PROGRAM TimeOptimizeCtrl
VAR
(************************ MinMax Declaration  *********************************************************************************)
	fbV2MasterTimeBlockWithMinMax: fbV2_MasterTimeBlockWithMinMax;
	LDBasketInfo: DSV2_BasketInfo;

	AR3SiSortedMTBFreeArm_Scanning				: ARRAY[1..iArmQty, 1..iMasterBlockQty, 1..3] OF INT;
	AR3SiSortedMTBFreeStn_Scanning				: ARRAY[1..iStnQty, 1..iMasterBlockQty, 1..3] OF INT;
	AR3SiSortedMTBFreeUld_Scanning				: ARRAY[1..iUldStnQty, 1..iMasterBlockQty, 1..3] OF INT;
	ARiMTBFreeSlotDataQtyArm_Scanning			: ARRAY[1..iArmQty] OF INT;
	ARiMTBFreeSlotDataQtyStn_Scanning			: ARRAY[1..iStnQty] OF INT;
	ARiMTBFreeSlotDataQtyUld_Scanning			: ARRAY[1..iUldStnQty] OF INT;

	bScanBusyFlag						: BOOL;

	diSinceStartRunningTime					: DINT;
	diSinceCopyRunningTime					: DINT;
	iCheckStep								: INT;
	bAutoRetry								: BOOL;
	tAutoRetryTimerEV						: TIME;



(************************ MinMax Declaration END *********************************************************************************)



	DelayTime: TIME := t#1s;
	TON2: TON;
	LdPnpStRE: R_TRIG;
	LdPnpStFE: F_TRIG;



	bManualRecipeGenerateEN: BOOL;
(*	fbV2SubMTBFreeSlotGenerator: fbV2_SubMTBFreeSlotGenerator;*)
	MTB_ArmTimeOK: BOOL;
	ArmPnpStep3: BOOL;
	bArmPnpStep3: BOOL;
	bArmPnpStep5: BOOL;
END_VAR

VAR PERSISTENT

	AR2SiManualSimulationInput : ARRAY [1..iRecipeBlockQty, 1..2] OF INT;  (*1st Array=Steps 	2nd Array[1]=ProcessTime/ArmTransferTime 	2ndArray[2]=StnID*)
(*	AR2SiManualRecipeTimeBlockNoCallArmTime : ARRAY[1..iRecipeBlockQty, 1..3] OF INT;
	AR2SiManualRecipeTimeBlockWithCallArmTime : ARRAY[1..iRecipeBlockQty, 1..3] OF INT;
*)

(*	bSMTBFSG: BOOL;
	bBusy: BOOL;
	bDone : BOOL;
	ARiFreeSlotDataQtyArm									: ARRAY[1..iArmQty] OF INT;
	ARiFreeSlotDataQtyStn									: ARRAY[1..iStnQty] OF INT;
	ARiFreeSlotDataQtyUld									: ARRAY[1..iUldStnQty] OF INT;


	AR3SiMasterTimeBlockFreeArm_MTB		 			: ARRAY[1..iArmQty, 1..iMasterBlockQty, 1..3] OF INT;
	AR3SiMasterTimeBlockFreeStn_MTB					: ARRAY[1..iStnQty, 1..iMasterBlockQty, 1..3] OF INT;
	AR3SiMasterTimeBlockFreeUld_MTB					: ARRAY[1..iUldStnQty, 1..iMasterBlockQty, 1..3] OF INT;
*)
END_VAR

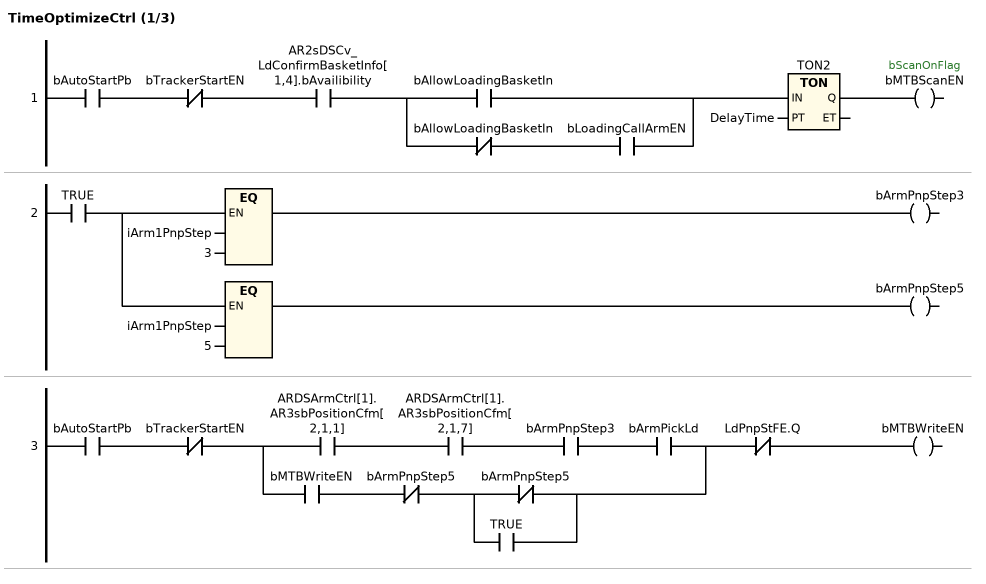
// NETWORK 1
//   bMTBScanEN: bScanOnFlag
TON2(IN := bAutoStartPb AND NOT bTrackerStartEN AND AR2sDSCv_LdConfirmBasketInfo[1,4].bAvailibility AND (bAllowLoadingBasketIn OR NOT bAllowLoadingBasketIn AND bLoadingCallArmEN), PT := DelayTime); // TON
bMTBScanEN := TON2.Q;

// NETWORK 2
bArmPnpStep3 := iArm1PnpStep = 3;
bArmPnpStep5 := iArm1PnpStep = 5;

// NETWORK 3
bMTBWriteEN := (bAutoStartPb AND NOT bTrackerStartEN AND (ARDSArmCtrl[1].AR3sbPositionCfm[2,1,1] AND ARDSArmCtrl[1].AR3sbPositionCfm[2,1,7] AND bArmPnpStep3 AND bArmPickLd OR bMTBWriteEN AND NOT bArmPnpStep5 AND (NOT bArmPnpStep5 OR TRUE))) AND NOT LdPnpStFE.Q;

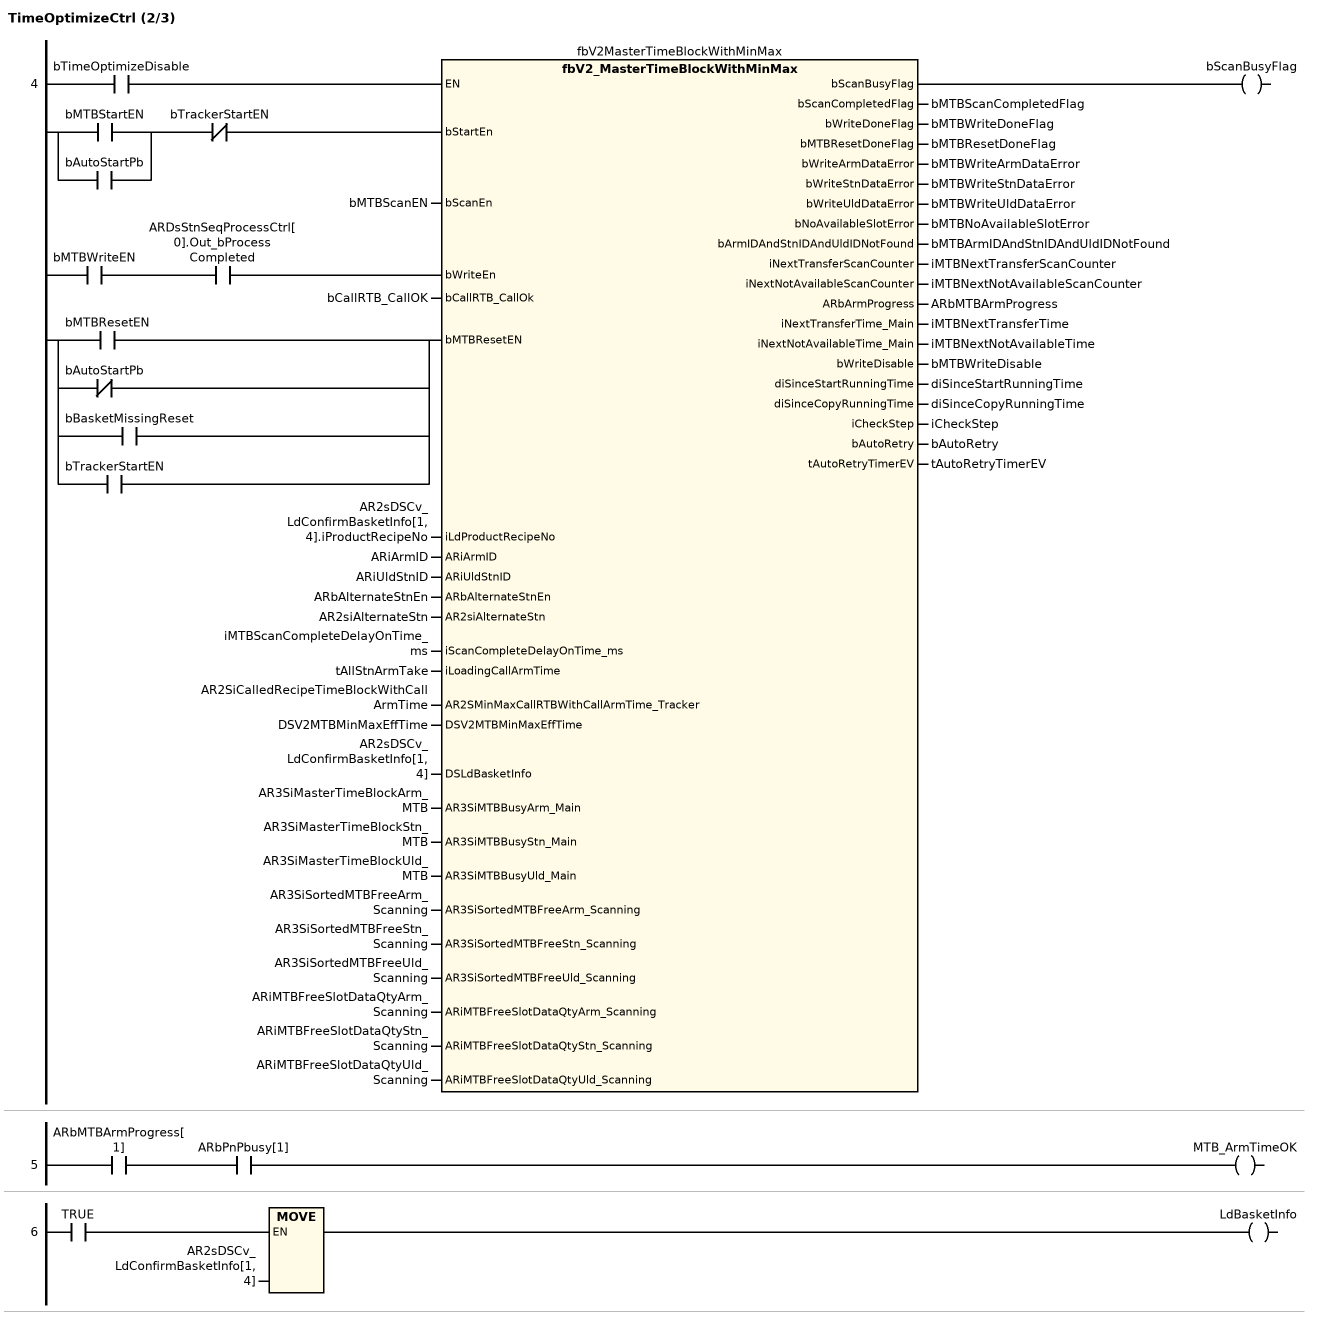
// NETWORK 4
IF bTimeOptimizeDisable THEN
    fbV2MasterTimeBlockWithMinMax(
        bStartEn := (bMTBStartEN OR bAutoStartPb) AND NOT bTrackerStartEN,
        bScanEn := bMTBScanEN,
        bWriteEn := bMTBWriteEN AND ARDsStnSeqProcessCtrl[0].Out_bProcessCompleted,
        bCallRTB_CallOk := bCallRTB_CallOK,
        bMTBResetEN := bMTBResetEN OR NOT bAutoStartPb OR bBasketMissingReset OR bTrackerStartEN,
        iLdProductRecipeNo := AR2sDSCv_LdConfirmBasketInfo[1,4].iProductRecipeNo,
        ARiArmID := ARiArmID,
        ARiUldStnID := ARiUldStnID,
        ARbAlternateStnEn := ARbAlternateStnEn,
        AR2siAlternateStn := AR2siAlternateStn,
        iScanCompleteDelayOnTime_ms := iMTBScanCompleteDelayOnTime_ms,
        iLoadingCallArmTime := tAllStnArmTake,
        AR2SMinMaxCallRTBWithCallArmTime_Tracker := AR2SiCalledRecipeTimeBlockWithCallArmTime,
        DSV2MTBMinMaxEffTime := DSV2MTBMinMaxEffTime,
        DSLdBasketInfo := AR2sDSCv_LdConfirmBasketInfo[1,4],
        AR3SiMTBBusyArm_Main := AR3SiMasterTimeBlockArm_MTB,
        AR3SiMTBBusyStn_Main := AR3SiMasterTimeBlockStn_MTB,
        AR3SiMTBBusyUld_Main := AR3SiMasterTimeBlockUld_MTB,
        AR3SiSortedMTBFreeArm_Scanning := AR3SiSortedMTBFreeArm_Scanning,
        AR3SiSortedMTBFreeStn_Scanning := AR3SiSortedMTBFreeStn_Scanning,
        AR3SiSortedMTBFreeUld_Scanning := AR3SiSortedMTBFreeUld_Scanning,
        ARiMTBFreeSlotDataQtyArm_Scanning := ARiMTBFreeSlotDataQtyArm_Scanning,
        ARiMTBFreeSlotDataQtyStn_Scanning := ARiMTBFreeSlotDataQtyStn_Scanning,
        ARiMTBFreeSlotDataQtyUld_Scanning := ARiMTBFreeSlotDataQtyUld_Scanning,
        bScanCompletedFlag => bMTBScanCompletedFlag,
        bWriteDoneFlag => bMTBWriteDoneFlag,
        bMTBResetDoneFlag => bMTBResetDoneFlag,
        bWriteArmDataError => bMTBWriteArmDataError,
        bWriteStnDataError => bMTBWriteStnDataError,
        bWriteUldDataError => bMTBWriteUldDataError,
        bNoAvailableSlotError => bMTBNoAvailableSlotError,
        bArmIDAndStnIDAndUldIDNotFound => bMTBArmIDAndStnIDAndUldIDNotFound,
        iNextTransferScanCounter => iMTBNextTransferScanCounter,
        iNextNotAvailableScanCounter => iMTBNextNotAvailableScanCounter,
        ARbArmProgress => ARbMTBArmProgress,
        iNextTransferTime_Main => iMTBNextTransferTime,
        iNextNotAvailableTime_Main => iMTBNextNotAvailableTime,
        bWriteDisable => bMTBWriteDisable,
        diSinceStartRunningTime => diSinceStartRunningTime,
        diSinceCopyRunningTime => diSinceCopyRunningTime,
        iCheckStep => iCheckStep,
        bAutoRetry => bAutoRetry,
        tAutoRetryTimerEV => tAutoRetryTimerEV); // fbV2_MasterTimeBlockWithMinMax
END_IF
bScanBusyFlag := fbV2MasterTimeBlockWithMinMax.bScanBusyFlag;

// NETWORK 5
MTB_ArmTimeOK := ARbMTBArmProgress[1] AND ARbPnPbusy[1];

// NETWORK 6
LdBasketInfo := AR2sDSCv_LdConfirmBasketInfo[1,4];

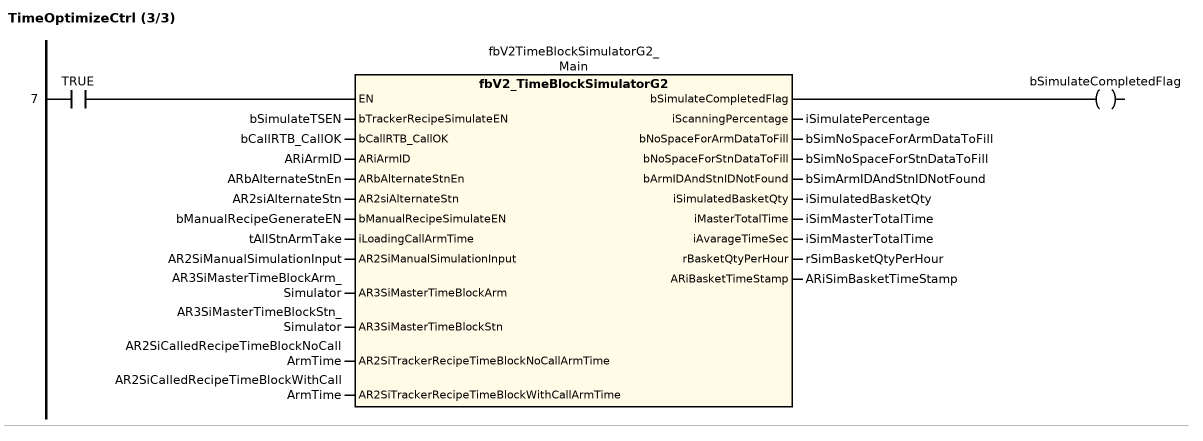
// NETWORK 7
fbV2TimeBlockSimulatorG2_Main(
    bTrackerRecipeSimulateEN := bSimulateTSEN,
    bCallRTB_CallOK := bCallRTB_CallOK,
    ARiArmID := ARiArmID,
    ARbAlternateStnEn := ARbAlternateStnEn,
    AR2siAlternateStn := AR2siAlternateStn,
    bManualRecipeSimulateEN := bManualRecipeGenerateEN,
    iLoadingCallArmTime := tAllStnArmTake,
    AR2SiManualSimulationInput := AR2SiManualSimulationInput,
    AR3SiMasterTimeBlockArm := AR3SiMasterTimeBlockArm_Simulator,
    AR3SiMasterTimeBlockStn := AR3SiMasterTimeBlockStn_Simulator,
    AR2SiTrackerRecipeTimeBlockNoCallArmTime := AR2SiCalledRecipeTimeBlockNoCallArmTime,
    AR2SiTrackerRecipeTimeBlockWithCallArmTime := AR2SiCalledRecipeTimeBlockWithCallArmTime,
    iScanningPercentage => iSimulatePercentage,
    bNoSpaceForArmDataToFill => bSimNoSpaceForArmDataToFill,
    bNoSpaceForStnDataToFill => bSimNoSpaceForStnDataToFill,
    bArmIDAndStnIDNotFound => bSimArmIDAndStnIDNotFound,
    iSimulatedBasketQty => iSimulatedBasketQty,
    iMasterTotalTime => iSimMasterTotalTime,
    iAvarageTimeSec => iSimMasterTotalTime,
    rBasketQtyPerHour => rSimBasketQtyPerHour,
    ARiBasketTimeStamp => ARiSimBasketTimeStamp); // fbV2_TimeBlockSimulatorG2
bSimulateCompletedFlag := fbV2TimeBlockSimulatorG2_Main.bSimulateCompletedFlag;

END_PROGRAM

(* stored: Version 1.1.0.1, ProductVersion 3.1.4024.12
   POU TimeOptimizeCtrl: Id {a002940d-fddb-4e48-ac33-87202f706f04}, SpecialFunc None *)
